// TIA Portal project "Prueba_ODK_DialogBox" (V16)

(* hardware
DEVICE "S71500/ET200MP station_1"  S7-1500 station
   slot 0: "Rail_0"  Rack  6ES7 590-1***0-0AA0
   slot 1: "PLC_1"  CPU 1518-4 PN/DP  6ES7 518-4AP00-3AB0  V2.8
      slot 3: "CPU display_1"  6ES7591-1BA00-0AA0
      slot 32768: "PROFINET interface_1"  X1
         slot 32769: "Port_1"  X1 P1
         slot 32770: "Port_2"  X1 P2
      slot 33024: "PROFINET interface_2"  X2
         slot 33025: "Port_1"  X2 P1
      slot 33280: "PROFINET interface GBIT_3"  X3
         slot 33281: "Port_1"  X3 P1
      slot 33536: "DP interface_1"  X4
      slot 34817: "Virtual CP interface port_1"  Virtual CP interface port  Virtual CP interface port
*)

// ===== PLC "PLC_1"  CPU 1518-4 PN/DP =====

VAR_GLOBAL   // PLC tag table "Default tag table"
   "Tag_1" AT %M0.0 : Bool;
END_VAR

TYPE "ODKProject7control_flags"
// This block is AUTO GENERATED - DO NOT MODIFY this block!
// Created by ODK_CodeGenerator version 205.100.101.18
// at Thu December 3 18:06:44 2020
// ********************************************************
   STRUCT
      Control_Flag_New_Service : Bool;
      Control_Flag_Item_Completed : Bool;
      Control_Flag_Service_Completed : Bool;
   END_STRUCT;
END_TYPE

TYPE "ODKProject7agent2plc"
// This block is AUTO GENERATED - DO NOT MODIFY this block!
// Created by ODK_CodeGenerator version 205.100.101.18
// at Thu December 3 18:06:44 2020
// ********************************************************
   STRUCT
      Id_Machine_Reference : UDInt;
      Id_Order_Reference : UDInt;
      Id_Batch_Reference : UDInt;
      Id_Ref_Subproduct_Type : UDInt;
      Operation_Ref_Service_Type : UDInt;
      Operation_No_of_Items : USInt;
   END_STRUCT;
END_TYPE

TYPE "ODKProject7plc2agent"
// This block is AUTO GENERATED - DO NOT MODIFY this block!
// Created by ODK_CodeGenerator version 205.100.101.18
// at Thu December 3 18:06:44 2020
// ********************************************************
   STRUCT
      Id_Machine_Reference : UDInt;
      Id_Order_Reference : UDInt;
      Id_Batch_Reference : UDInt;
      Id_Ref_Subproduct_Type : UDInt;
      Id_Ref_Service_Type : UDInt;
      Id_Item_Number : USInt;
      Data_Initial_Time_Stamp : LDT;
      Data_Final_Time_Stamp : LDT;
      Data_Service_Time_Stamp : LDT;
   END_STRUCT;
END_TYPE

TYPE "agent2plc"
   STRUCT
      Id_Machine_Reference : UDInt;
      Id_Order_Reference : UDInt;
      Id_Batch_Reference : UDInt;
      Id_Ref_Subproduct_Type : UDInt;
      Operation_Ref_Service_Type : UDInt;
      Operation_No_of_Items : USInt;
   END_STRUCT;
END_TYPE

TYPE "ODKProject2control_flags"
// This block is AUTO GENERATED - DO NOT MODIFY this block!
// Created by ODK_CodeGenerator version 205.100.101.18
// at Wed December 9 10:48:10 2020
// ********************************************************
   STRUCT
      Control_Flag_New_Service : Bool;
      Control_Flag_Item_Completed : Bool;
      Control_Flag_Service_Completed : Bool;
   END_STRUCT;
END_TYPE

TYPE "ODKProject2agent2plc"
// This block is AUTO GENERATED - DO NOT MODIFY this block!
// Created by ODK_CodeGenerator version 205.100.101.18
// at Wed December 9 10:48:10 2020
// ********************************************************
   STRUCT
      Id_Machine_Reference : UDInt;
      Id_Order_Reference : UDInt;
      Id_Batch_Reference : UDInt;
      Id_Ref_Subproduct_Type : UDInt;
      Operation_Ref_Service_Type : UDInt;
      Operation_No_of_Items : USInt;
   END_STRUCT;
END_TYPE

TYPE "ODKProject2plc2agent"
// This block is AUTO GENERATED - DO NOT MODIFY this block!
// Created by ODK_CodeGenerator version 205.100.101.18
// at Wed December 9 10:48:10 2020
// ********************************************************
   STRUCT
      Id_Machine_Reference : UDInt;
      Id_Order_Reference : UDInt;
      Id_Batch_Reference : UDInt;
      Id_Ref_Subproduct_Type : UDInt;
      Id_Ref_Service_Type : UDInt;
      Id_Item_Number : USInt;
      Data_Initial_Time_Stamp : LDT;
      Data_Final_Time_Stamp : LDT;
      Data_Service_Time_Stamp : LDT;
   END_STRUCT;
END_TYPE

DATA_BLOCK "ODKProject1Publish_DB"   // DB1
{ S7_Optimized_Access := 'TRUE' }
VERSION : 0.1
// stored: InstanceOfName ODKProject1Publish
"ODKProject1Publish"
BEGIN
END_DATA_BLOCK

DATA_BLOCK "ODKProject1CheckSubscriptions_DB"   // DB2
{ S7_Optimized_Access := 'TRUE' }
VERSION : 0.1
// stored: InstanceOfName ODKProject1CheckSubscriptions
"ODKProject1CheckSubscriptions"
BEGIN
END_DATA_BLOCK

DATA_BLOCK "ODKProject1_Unload_DB"   // DB3
{ S7_Optimized_Access := 'TRUE' }
VERSION : 0.1
// stored: InstanceOfName ODKProject1_Unload
"ODKProject1_Unload"
BEGIN
END_DATA_BLOCK

DATA_BLOCK "ODK_function_DB"   // DB4
{ S7_Optimized_Access := 'TRUE' }
VERSION : 0.1
   VAR
      load_Function : Bool := false;
      unload_Function : Bool;
      mensaje : String := 'Kaixo!';
      publicar : Bool;
   END_VAR
BEGIN
END_DATA_BLOCK

DATA_BLOCK "ODKProject1_GetTrace_DB"   // DB5
{ S7_Optimized_Access := 'TRUE' }
VERSION : 0.1
// stored: InstanceOfName ODKProject1_GetTrace
"ODKProject1_GetTrace"
BEGIN
END_DATA_BLOCK

DATA_BLOCK "ODKProject1_Load_DB"   // DB6
{ S7_Optimized_Access := 'TRUE' }
VERSION : 0.1
// stored: InstanceOfName ODKProject1_Load
"ODKProject1_Load"
BEGIN
END_DATA_BLOCK

FUNCTION_BLOCK "ODKProject1_Load"   // FB1, SCL
{ S7_Optimized_Access := 'TRUE' }
VERSION : 0.1
// This block is AUTO GENERATED - DO NOT MODIFY this block!
// Created by ODK_CodeGenerator version 2.5.1
// at Sun June 19 23:40:51 2022
// max. number of parallel calls into this ODK application is: 3
// *************************************************************
   VAR_INPUT
      REQ : Bool;
   END_VAR
   VAR_OUTPUT
      DONE : Bool;
      BUSY : Bool;
      ERROR : Bool;
      STATUS : Int;
   END_VAR
   VAR
      ODK_Load_Instance : ODK_Load;
      _odk_internal_LIBRARY_NAME : String := '<rt>ODKProject1.dll';
   END_VAR
   VAR CONSTANT
      _odk_internal_INSTANCE_ID : UDInt := 993_767_873;
   END_VAR
BEGIN
   //
   // DO NOT CHANGE BELOW OF THIS LINE !!
   // This is an automatic generated block by the
   // SIMATIC ODK 1500S V2.5.1
   // DO NOT CHANGE !!
   //
   #ODK_Load_Instance(REQ := #REQ,
                      LIBRARY_NAME := #_odk_internal_LIBRARY_NAME,
                      INSTANCE_ID := #_odk_internal_INSTANCE_ID,
                      DONE => #DONE,
                      BUSY => #BUSY,
                      ERROR => #ERROR,
                      STATUS => #STATUS);
   //
   // DO NOT CHANGE !!
   // This is an automatic generated block by the
   // SIMATIC ODK 1500S V2.5.1
   // DO NOT CHANGE ABOVE OF THIS LINE !!
   //
END_FUNCTION_BLOCK

FUNCTION_BLOCK "ODKProject1_Unload"   // FB2, SCL
{ S7_Optimized_Access := 'TRUE' }
VERSION : 0.1
// This block is AUTO GENERATED - DO NOT MODIFY this block!
// Created by ODK_CodeGenerator version 205.100.101.18
// at Sun June 19 23:40:51 2022
// max. number of parallel calls into this ODK application is: 3
// *************************************************************
   VAR_INPUT
      REQ : Bool;
   END_VAR
   VAR_OUTPUT
      DONE : Bool;
      BUSY : Bool;
      ERROR : Bool;
      STATUS : Int;
   END_VAR
   VAR
      ODK_Unld_Instance : ODK_Unld;
   END_VAR
   VAR CONSTANT
      _odk_internal_INSTANCE_ID : UDInt := 993_767_873;
   END_VAR
BEGIN
   //
   // DO NOT CHANGE BELOW OF THIS LINE !!
   // This is an automatic generated block by the
   // SIMATIC ODK 1500S V2.5.1
   // DO NOT CHANGE !!
   //
   #ODK_Unld_Instance(REQ := #REQ,
                      INSTANCE_ID := #_odk_internal_INSTANCE_ID,
                      DONE => #DONE,
                      BUSY => #BUSY,
                      ERROR => #ERROR,
                      STATUS => #STATUS);
   //
   // DO NOT CHANGE !!
   // This is an automatic generated block by the
   // SIMATIC ODK 1500S V2.5.1
   // DO NOT CHANGE ABOVE OF THIS LINE !!
   //
END_FUNCTION_BLOCK

FUNCTION_BLOCK "ODKProject1Publish"   // FB3, SCL
{ S7_Optimized_Access := 'TRUE' }
VERSION : 0.1
// This block is AUTO GENERATED - DO NOT MODIFY this block!
// Created by ODK_CodeGenerator version 205.100.101.18
// at Sun June 19 23:40:51 2022
// max. number of parallel calls into this ODK application is: 3
// *************************************************************
//  Basic function in order to show 
//  how to create a function in ODK 1500S.
   VAR_INPUT
      message : String[254];
   END_VAR
   VAR_OUTPUT
      STATUS : Int := 0;
   END_VAR
   VAR
      _odk_internal_Last_REQ : Bool := FALSE;
      _odk_internal_Last_BUSY : Bool := FALSE;
      _odk_internal_IN_BUFFER : Array[0..255] of Byte;
   END_VAR
   VAR_TEMP
      _odk_internal_pos : DInt;
      _odk_internal_err : Int;
      _odk_internal_i : Int;
      _odk_internal_tmpStringLen : Byte;
   END_VAR
   VAR CONSTANT
      _odk_internal_INSTANCE_ID : UDInt := 993_767_873;
      _odk_internal_COMMAND : UDInt := 733_636_168;
   END_VAR
BEGIN
   //
   // DO NOT CHANGE BELOW OF THIS LINE !!
   // This is an automatic generated block by the
   // SIMATIC ODK 1500S V2.5.1
   // DO NOT CHANGE !!
   //
   // Basic function in order to show 
   // how to create a function in ODK 1500S.
   #_odk_internal_pos := 0;
   #_odk_internal_tmpStringLen := INT_TO_BYTE(LEN(#message));
   #_odk_internal_IN_BUFFER[#_odk_internal_pos] := BYTE#254;
   #_odk_internal_pos := #_odk_internal_pos + 1;
   #_odk_internal_IN_BUFFER[#_odk_internal_pos] := #_odk_internal_tmpStringLen;
   #_odk_internal_pos := #_odk_internal_pos + 1;
   FOR #_odk_internal_i := 1 TO BYTE_TO_INT(#_odk_internal_tmpStringLen) DO
       #_odk_internal_IN_BUFFER[#_odk_internal_pos] := CHAR_TO_BYTE(#message[#_odk_internal_i]);
       #_odk_internal_pos := #_odk_internal_pos + 1;
   END_FOR;
   #_odk_internal_pos := #_odk_internal_pos + 254 - #_odk_internal_tmpStringLen;
   #STATUS := ODK_ExcS(INSTANCE_ID := #_odk_internal_INSTANCE_ID,
                       COMMAND := #_odk_internal_COMMAND,
                       IN_DATA := #_odk_internal_IN_BUFFER,
                       INOUT_DATA := null,
                       OUT_DATA := null);
   //
   // DO NOT CHANGE !!
   // This is an automatic generated block by the
   // SIMATIC ODK 1500S V2.5.1
   // DO NOT CHANGE ABOVE OF THIS LINE !!
   //
END_FUNCTION_BLOCK

FUNCTION_BLOCK "ODKProject1CheckSubscriptions"   // FB4, SCL
{ S7_Optimized_Access := 'TRUE' }
VERSION : 0.1
// This block is AUTO GENERATED - DO NOT MODIFY this block!
// Created by ODK_CodeGenerator version 205.100.101.18
// at Sun June 19 23:40:51 2022
// max. number of parallel calls into this ODK application is: 3
// *************************************************************
   VAR_OUTPUT
      STATUS : Int := 0;
      app2PLCtopic : String[254];
      app2PLCtopicLen : SInt;
      app2PLCmsg : String[254];
      app2PLCmsgLen : SInt;
   END_VAR
   VAR_IN_OUT
      flag : Bool;
   END_VAR
   VAR
      _odk_internal_Last_REQ : Bool := FALSE;
      _odk_internal_Last_BUSY : Bool := FALSE;
      _odk_internal_INOUT_BUFFER : Array[0..0] of Byte;
      _odk_internal_OUT_BUFFER : Array[0..513] of Byte;
   END_VAR
   VAR_TEMP
      _odk_internal_pos : DInt;
      _odk_internal_err : Int;
      _odk_internal_i : Int;
      _odk_internal_tmpStringLen : Byte;
   END_VAR
   VAR CONSTANT
      _odk_internal_INSTANCE_ID : UDInt := 993_767_873;
      _odk_internal_COMMAND : UDInt := 2_233_883_005;
   END_VAR
BEGIN
   //
   // DO NOT CHANGE BELOW OF THIS LINE !!
   // This is an automatic generated block by the
   // SIMATIC ODK 1500S V2.5.1
   // DO NOT CHANGE !!
   //
   #_odk_internal_pos := 0;
   IF (True = #flag) THEN
       #_odk_internal_INOUT_BUFFER[#_odk_internal_pos] := BYTE#1;
   ELSE
       #_odk_internal_INOUT_BUFFER[#_odk_internal_pos] := BYTE#0;
   END_IF;
   #_odk_internal_pos := #_odk_internal_pos + 1;
   #STATUS := ODK_ExcS(INSTANCE_ID := #_odk_internal_INSTANCE_ID,
                       COMMAND := #_odk_internal_COMMAND,
                       IN_DATA := null,
                       INOUT_DATA := #_odk_internal_INOUT_BUFFER,
                       OUT_DATA := #_odk_internal_OUT_BUFFER
   );
   IF INT_TO_UINT(#STATUS) < 16#7000 THEN
       #_odk_internal_pos := 0;
       #flag := BYTE_TO_BOOL(#_odk_internal_INOUT_BUFFER[#_odk_internal_pos]);
       #_odk_internal_pos := #_odk_internal_pos + 1;
       #_odk_internal_pos := 0;
       #app2PLCtopic := '';
       #_odk_internal_tmpStringLen := #_odk_internal_OUT_BUFFER[#_odk_internal_pos];
       #_odk_internal_pos := #_odk_internal_pos + 1;
       #_odk_internal_tmpStringLen := #_odk_internal_OUT_BUFFER[#_odk_internal_pos];
       #_odk_internal_pos := #_odk_internal_pos + 1;
       IF (254 < #_odk_internal_tmpStringLen) THEN
           #_odk_internal_tmpStringLen := 254;
       END_IF;
       FOR #_odk_internal_i := 1 TO BYTE_TO_INT(#_odk_internal_tmpStringLen) DO
           #app2PLCtopic[#_odk_internal_i] := BYTE_TO_CHAR(#_odk_internal_OUT_BUFFER[#_odk_internal_pos]);
           #_odk_internal_pos := #_odk_internal_pos + 1;
       END_FOR;
       #_odk_internal_pos := #_odk_internal_pos + 254 - LEN(#app2PLCtopic);
       #app2PLCtopicLen := BYTE_TO_SINT(#_odk_internal_OUT_BUFFER[#_odk_internal_pos]);
       #_odk_internal_pos := #_odk_internal_pos + 1;
       #app2PLCmsg := '';
       #_odk_internal_tmpStringLen := #_odk_internal_OUT_BUFFER[#_odk_internal_pos];
       #_odk_internal_pos := #_odk_internal_pos + 1;
       #_odk_internal_tmpStringLen := #_odk_internal_OUT_BUFFER[#_odk_internal_pos];
       #_odk_internal_pos := #_odk_internal_pos + 1;
       IF (254 < #_odk_internal_tmpStringLen) THEN
           #_odk_internal_tmpStringLen := 254;
       END_IF;
       FOR #_odk_internal_i := 1 TO BYTE_TO_INT(#_odk_internal_tmpStringLen) DO
           #app2PLCmsg[#_odk_internal_i] := BYTE_TO_CHAR(#_odk_internal_OUT_BUFFER[#_odk_internal_pos]);
           #_odk_internal_pos := #_odk_internal_pos + 1;
       END_FOR;
       #_odk_internal_pos := #_odk_internal_pos + 254 - LEN(#app2PLCmsg);
       #app2PLCmsgLen := BYTE_TO_SINT(#_odk_internal_OUT_BUFFER[#_odk_internal_pos]);
       #_odk_internal_pos := #_odk_internal_pos + 1;
   END_IF;
   //
   // DO NOT CHANGE !!
   // This is an automatic generated block by the
   // SIMATIC ODK 1500S V2.5.1
   // DO NOT CHANGE ABOVE OF THIS LINE !!
   //
END_FUNCTION_BLOCK

FUNCTION_BLOCK "ODKProject1_GetTrace"   // FB5, SCL
{ S7_Optimized_Access := 'TRUE' }
VERSION : 0.1
// This block is AUTO GENERATED - DO NOT MODIFY this block!
// Created by ODK_CodeGenerator version 205.100.101.18
// at Sun June 19 23:40:51 2022
// max. number of parallel calls into this ODK application is: 3
// *************************************************************
   VAR_INPUT
      TraceCount : Int;
   END_VAR
   VAR_OUTPUT
      STATUS : Int := 0;
      TraceBuffer : Array[0..255] of String[125];
   END_VAR
   VAR
      _odk_internal_Last_REQ : Bool := FALSE;
      _odk_internal_Last_BUSY : Bool := FALSE;
      _odk_internal_IN_BUFFER : Array[0..1] of Byte;
      _odk_internal_OUT_BUFFER : Array[0..32511] of Byte;
   END_VAR
   VAR_TEMP
      _odk_internal_pos : DInt;
      _odk_internal_err : Int;
      _odk_internal_i : Int;
      _odk_internal_tmpStringLen : Byte;
      _odk_internal_j : Int;
      _odk_internal_tmp_string : String;
   END_VAR
   VAR CONSTANT
      _odk_internal_INSTANCE_ID : UDInt := 993_767_873;
      _odk_internal_COMMAND : UDInt := 4_033_566_251;
   END_VAR
BEGIN
   //
   // DO NOT CHANGE BELOW OF THIS LINE !!
   // This is an automatic generated block by the
   // SIMATIC ODK 1500S V2.5.1
   // DO NOT CHANGE !!
   //
   #_odk_internal_pos := 0;
   #_odk_internal_err := WRITE_LITTLE(src_variable := #TraceCount, dest_array := #_odk_internal_IN_BUFFER, pos := #_odk_internal_pos);
   #STATUS := ODK_ExcS(INSTANCE_ID := #_odk_internal_INSTANCE_ID,
                       COMMAND := #_odk_internal_COMMAND,
                       IN_DATA := #_odk_internal_IN_BUFFER,
                       INOUT_DATA := null,
                       OUT_DATA := #_odk_internal_OUT_BUFFER
   );
   IF INT_TO_UINT(#STATUS) < 16#7000 THEN
       #_odk_internal_pos := 0;
       FOR #_odk_internal_j := 0 TO 255 DO
           #_odk_internal_tmp_string := '';
           #_odk_internal_tmpStringLen := #_odk_internal_OUT_BUFFER[#_odk_internal_pos];
           #_odk_internal_pos := #_odk_internal_pos + 1;
           #_odk_internal_tmpStringLen := #_odk_internal_OUT_BUFFER[#_odk_internal_pos];
           #_odk_internal_pos := #_odk_internal_pos + 1;
           IF (125 < #_odk_internal_tmpStringLen) THEN
               #_odk_internal_tmpStringLen := 125;
           END_IF;
           FOR #_odk_internal_i := 1 TO BYTE_TO_INT(#_odk_internal_tmpStringLen) DO
               #_odk_internal_tmp_string[#_odk_internal_i] := BYTE_TO_CHAR(#_odk_internal_OUT_BUFFER[#_odk_internal_pos]);
               #_odk_internal_pos := #_odk_internal_pos + 1;
           END_FOR;
           #_odk_internal_pos := #_odk_internal_pos + 125 - LEN(#_odk_internal_tmp_string);
           #TraceBuffer[#_odk_internal_j] := #_odk_internal_tmp_string;
       END_FOR;
   END_IF;
   //
   // DO NOT CHANGE !!
   // This is an automatic generated block by the
   // SIMATIC ODK 1500S V2.5.1
   // DO NOT CHANGE ABOVE OF THIS LINE !!
   //
END_FUNCTION_BLOCK

ORGANIZATION_BLOCK "Main"   // OB1, LAD, ProgramCycle
TITLE = "Main Program Sweep (Cycle)"
{ S7_Optimized_Access := 'TRUE' }
VERSION : 0.1
   VAR_INPUT
      Initial_Call : Bool;   // Initial call of this OB
      Remanence : Bool;   // =True, if remanent data are available
   END_VAR
   VAR_TEMP   // added for the SCL form of the ladder/FBD networks
      _w1 : Bool;
   END_VAR
BEGIN

REGION Network 1
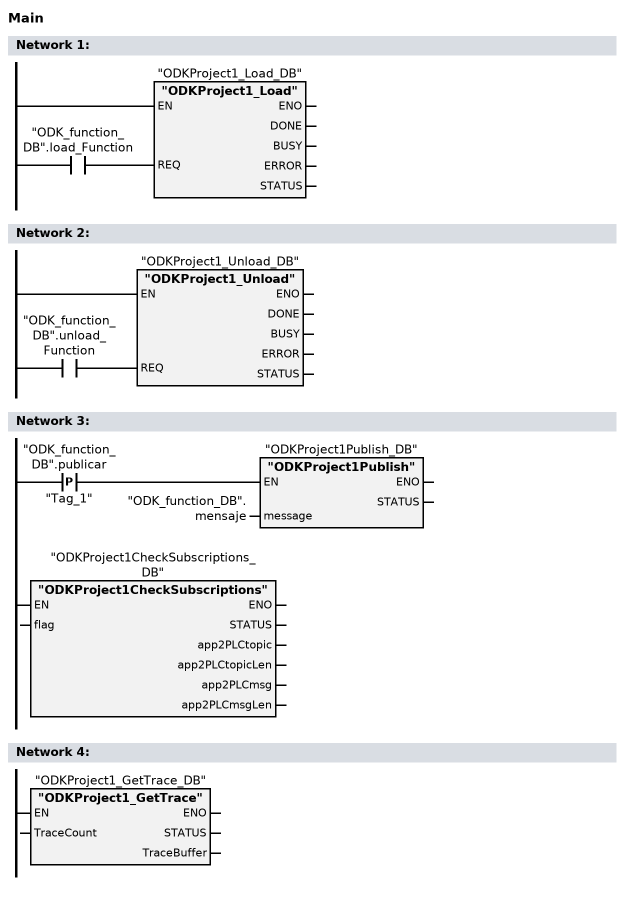
   RUNG wire#powerrail
      "ODKProject1_Load_DB"(REQ := wire#w1, DONE =>, BUSY =>, ERROR =>, STATUS =>)
   END_RUNG
   RUNG wire#powerrail
      Contact( "ODK_function_DB".load_Function )
   END_RUNG wire#w1
   // the same network as SCL:
   "ODKProject1_Load_DB"(REQ := "ODK_function_DB".load_Function);   // "ODKProject1_Load"
END_REGION

REGION Network 2
   RUNG wire#powerrail
      "ODKProject1_Unload_DB"(REQ := wire#w1, DONE =>, BUSY =>, ERROR =>, STATUS =>)
   END_RUNG
   RUNG wire#powerrail
      Contact( "ODK_function_DB".unload_Function )
   END_RUNG wire#w1
   // the same network as SCL:
   "ODKProject1_Unload_DB"(REQ := "ODK_function_DB".unload_Function);   // "ODKProject1_Unload"
END_REGION

REGION Network 3
   RUNG wire#powerrail
      P_Contact(operand := "ODK_function_DB".publicar, bit := "Tag_1")
      "ODKProject1Publish_DB"(message := "ODK_function_DB".mensaje, STATUS =>)
   END_RUNG
   RUNG wire#powerrail
      "ODKProject1CheckSubscriptions_DB"(flag :=, STATUS =>, app2PLCtopic =>, app2PLCtopicLen =>, app2PLCmsg =>, app2PLCmsgLen =>)
   END_RUNG
   // the same network as SCL:
   #_w1 := "ODK_function_DB".publicar AND NOT "Tag_1";   // rising edge of "ODK_function_DB".publicar
   "Tag_1" := "ODK_function_DB".publicar;
   IF #_w1 THEN
       "ODKProject1Publish_DB"(message := "ODK_function_DB".mensaje);   // "ODKProject1Publish"
   END_IF;
   "ODKProject1CheckSubscriptions_DB"();   // "ODKProject1CheckSubscriptions"
END_REGION

REGION Network 4
   RUNG wire#powerrail
      "ODKProject1_GetTrace_DB"(TraceCount :=, STATUS =>, TraceBuffer =>)
   END_RUNG
   // the same network as SCL:
   "ODKProject1_GetTrace_DB"();   // "ODKProject1_GetTrace"
END_REGION
END_ORGANIZATION_BLOCK